(* Logix 5000 project; controller SRP_BullPMM_TestBench_V1 vendor 1 type 14 code 77 rev 20.11; software revision 20.04 *)

TASK MainTask (continuous, watchdog 500 ms) : MainProgram

MODULES
   Controller : vendor 1 type 14 code 77 (CompactLogixL32EController 0, rev 20.11)
      LocalENB : 1769-L32E Ethernet Port (CompactLogixL32Ethernet 1, rev 20.11)
         VSD_DC : vendor 1 type 123 code 121 (Ethernet 192.168.2.130, rev 5.6, Output RPI 20 ms)
             : vendor 1 type 123 code 8192 (DPI 5, rev 4.1)
      Local : CompactBus (CompactVirtualAdapter 3, rev 20.11)
END_MODULES

VAR_GLOBAL   (* controller tags *)
   CTU_SRPSim : COUNTER := (PRE := 142, ACC := 32);
   DC_CommandOFF : BOOL;
   DC_CommandON : BOOL;
   DC_CommandReset : BOOL;
   DC_CommandSpeed : INT;
   DC_CurrentLimit : INT;
   DC_LoadSent : INT := 10;
   DC_MaxLoad : REAL := 15.0;
   DC_MinLoad : REAL := 3.0;
   DC_OutputPower : REAL;
   DC_OutputVoltage : REAL;
   DC_RPMFeedback : INT := -12;
   DC_RPMReference : DINT := -13;
   DC_SpeedReference : INT;
   DC_Timer_OFF : TIMER := (PRE := 1000);
   DC_Timer_ON : TIMER := (PRE := 1000);
   DC_Timer_RST : TIMER := (PRE := 1000);
   Samples : INT := 142;
   SPM : REAL := 8.51;
   SRP_MaxPower : REAL := 10.0;
   SRP_MinPower : REAL := -7.1723228;
   SRP_Power : REAL[400] := ([0] := 4.524285, [1] := 3.699268, [2] := 2.7944112, [3] := 2.3752496, [4] := 2.3020627, [5] := 1.8629409, [6] := 1.3023952, [7] := 0.87658024, [8] := 0.60296065, [9] := -0.33848965, [10] := -1.7365268, [11] := -1.9893546, [12] := -1.428809, [13] := -1.2059215, [14] := -1.8562874, [15] := -2.4950101, [16] := -2.5748503, [17] := -2.3353293, [18] := -2.2821023, [19] := -2.255489, [20] := -1.8829011, [21] := -1.2724552, [22] := -0.78925484, [23] := -0.57717896, [24] := -0.59713894, [25] := -0.6320692, [26] := -0.55056554, [27] := -0.42997342, [28] := -0.11747335, [29] := 0.09813703, [30] := 0.18099219, [31] := 0.5006655, [32] := 2.2089155, [33] := 3.8855622, [34] := 3.379907, [35] := 2.3885562, [36] := 1.9560877, [37] := 3.1536927, [38] := 4.23819, [39] := 4.0119762, [40] := 3.732535, [41] := 4.4777117, [42] := 5.3892217, [43] := 5.282768, [44] := 4.8835664, [45] := 5.269461, [46] := 5.9946775, [47] := 6.0745177, [48] := 5.974717, [49] := 6.5336, [50] := 7.3586164, [51] := 7.711244, [52] := 7.498337, [53] := 7.784431, [54] := 8.263473, [55] := 8.616101, [56] := 8.562874, [57] := 8.755822, [58] := 9.248171, [59] := 9.634065,
        [60] := 9.720559, [61] := 9.720559, [62] := 9.833667, [63] := 10.0, [64] := 9.893547, [65] := 9.720559, [66] := 9.713905, [67] := 9.680639, [68] := 9.414504, [69] := 9.161676, [70] := 9.161676, [71] := 9.061876, [72] := 8.576181, [73] := 8.190286, [74] := 8.097139, [75] := 7.837658, [76] := 7.3320026, [77] := 6.9194946, [78] := 6.69328, [79] := 6.267465, [80] := 5.6753163, [81] := 5.169661, [82] := 4.8103795, [83] := 4.4045243, [84] := 3.918829, [85] := 3.2601464, [86] := 2.7145708, [87] := 2.255489, [88] := 1.8030605, [89] := 1.318197, [90] := 0.9564206, [91] := 0.7202261, [92] := 0.50731874, [93] := -0.14678977, [94] := -2.1091151, [95] := -3.3399868, [96] := -3.2468398, [97] := -3.0139723, [98] := -3.7924154, [99] := -5.056554, [100] := -5.5688624, [101] := -5.482369, [102] := -5.788423, [103] := -6.600133, [104] := -7.0991354, [105] := -7.0725217, [106] := -7.019295, [107] := -7.1723228, [108] := -7.092482, [109] := -6.2208915, [110] := -5.1430473, [111] := -4.291417, [112] := -3.4464405, [113] := -2.1290753, [114] := -1.0703592, [115] := 1.7631403, [116] := 6.5934796, [117] := 8.243513, [118] := 6.6799736, [119] := 5.968064,
        [120] := 7.604791, [121] := 8.383234, [122] := 6.952761, [123] := 5.768463, [124] := 6.5735197, [125] := 7.458417, [126] := 6.759814, [127] := 5.449102, [128] := 5.475715, [129] := 6.1011314, [130] := 5.76181, [131] := 4.6240854, [132] := 4.770459, [133] := 5.9614105, [134] := 6.320692, [135] := 5.635396, [136] := 5.269461, [137] := 5.928144, [138] := 6.081171, [139] := 5.1297407, [140] := 4.3313375, [141] := 4.4444447);
   SRP_SimActualPower : REAL := 2.2089155;
   SRP_SimActualStroke : DINT; {produced}
   SRP_Simulation : BOOL := 1;
   SRP_StrokeDetection : INT[400] := ([0] := 1, [1] := 1, [2] := 1, [3] := 1, [4] := 1, [5] := 1, [6] := 1);
   Test_TagExcel : INT := 1;
   Timer_SRPsim : TIMER := (PRE := 50, ACC := 14, EN := 1, TT := 1);
END_VAR

PROGRAM MainProgram   (* main routine MainRoutine *)
VAR
   SCL_01 : SCALE := (In := 1.9560877, InRawMax := 10.0, InRawMin := -7.1723228, InEUMax := 15.0, InEUMin := 3.0, Out := 9.378923);
END_VAR

ROUTINE MainRoutine   (* ladder *)
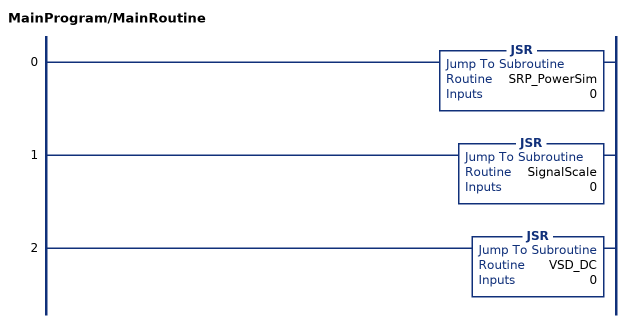
   0: JSR(SRP_PowerSim,0);
   1: JSR(SignalScale,0);
   2: JSR(VSD_DC,0);
END_ROUTINE

ROUTINE SignalScale   (* function block diagram *)
   SHEET 1
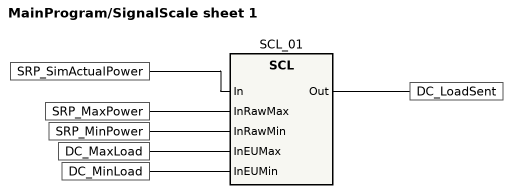
   SCL_01 : SCL(In := SRP_SimActualPower, InRawMax := SRP_MaxPower, InRawMin := SRP_MinPower, InEUMax := DC_MaxLoad, InEUMin := DC_MinLoad);
   DC_LoadSent := SCL_01.Out;
END_ROUTINE

ROUTINE SRP_PowerSim   (* ladder *)
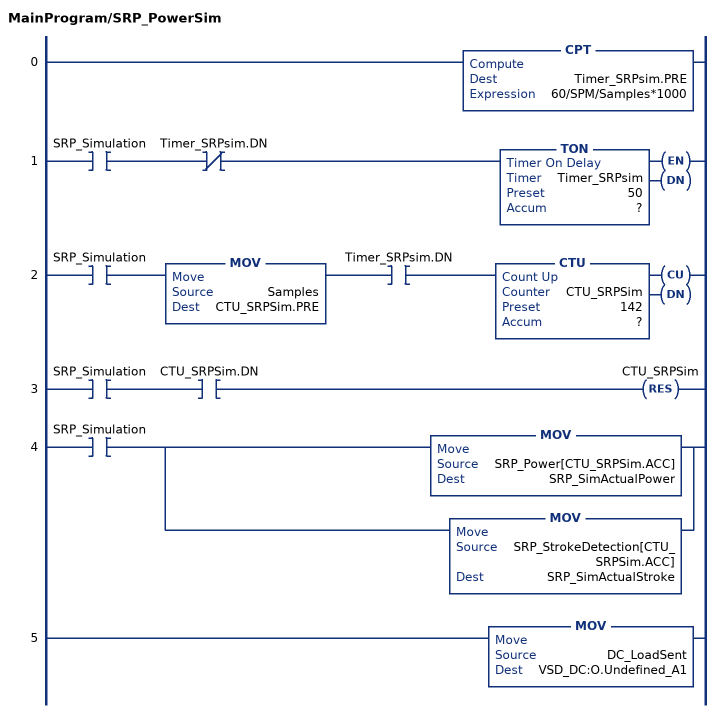
   0: CPT(Timer_SRPsim.PRE,60/SPM/Samples*1000);
   1: XIC(SRP_Simulation)XIO(Timer_SRPsim.DN)TON(Timer_SRPsim,?,?);
   2: XIC(SRP_Simulation)MOV(Samples,CTU_SRPSim.PRE)XIC(Timer_SRPsim.DN)CTU(CTU_SRPSim,?,?);
   3: XIC(SRP_Simulation)XIC(CTU_SRPSim.DN)RES(CTU_SRPSim);
   4: XIC(SRP_Simulation)[MOV(SRP_Power[CTU_SRPSim.ACC],SRP_SimActualPower) ,MOV(SRP_StrokeDetection[CTU_SRPSim.ACC],SRP_SimActualStroke) ];
   5: MOV(DC_LoadSent,VSD_DC:O.Undefined_A1);
END_ROUTINE

ROUTINE VSD_DC   (* ladder *)
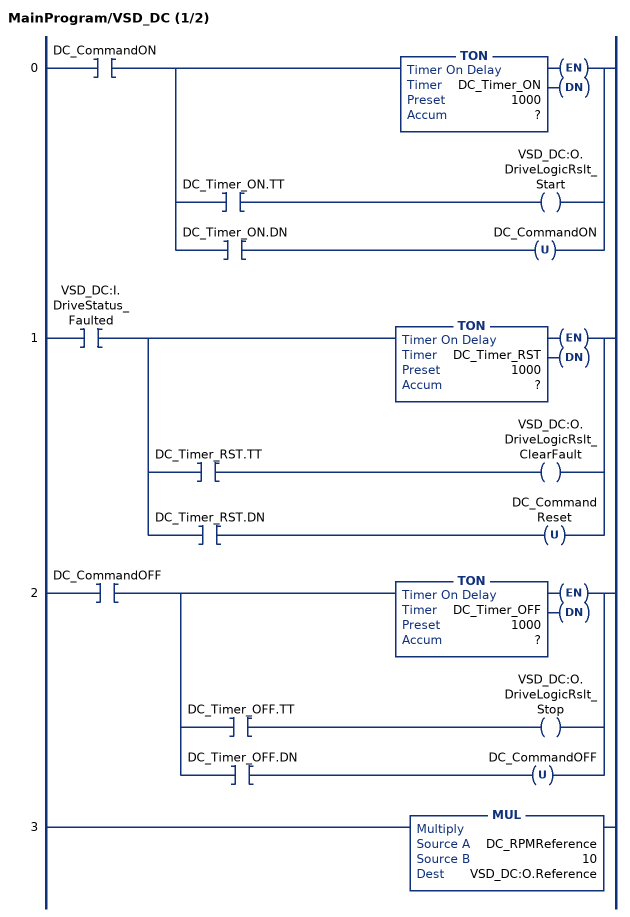
   0: XIC(DC_CommandON)[TON(DC_Timer_ON,?,?) ,[XIC(DC_Timer_ON.TT) OTE(VSD_DC:O.DriveLogicRslt_Start) ,XIC(DC_Timer_ON.DN) OTU(DC_CommandON) ] ];
   1: XIC(VSD_DC:I.DriveStatus_Faulted)[TON(DC_Timer_RST,?,?) ,[XIC(DC_Timer_RST.TT) OTE(VSD_DC:O.DriveLogicRslt_ClearFault) ,XIC(DC_Timer_RST.DN) OTU(DC_CommandReset) ] ];
   2: XIC(DC_CommandOFF)[TON(DC_Timer_OFF,?,?) ,[XIC(DC_Timer_OFF.TT) OTE(VSD_DC:O.DriveLogicRslt_Stop) ,XIC(DC_Timer_OFF.DN) OTU(DC_CommandOFF) ] ];
   3: MUL(DC_RPMReference,10,VSD_DC:O.Reference);
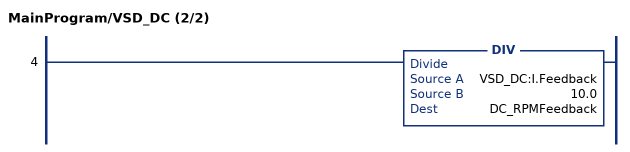
   4: DIV(VSD_DC:I.Feedback,10.0,DC_RPMFeedback);
END_ROUTINE
END_PROGRAM
